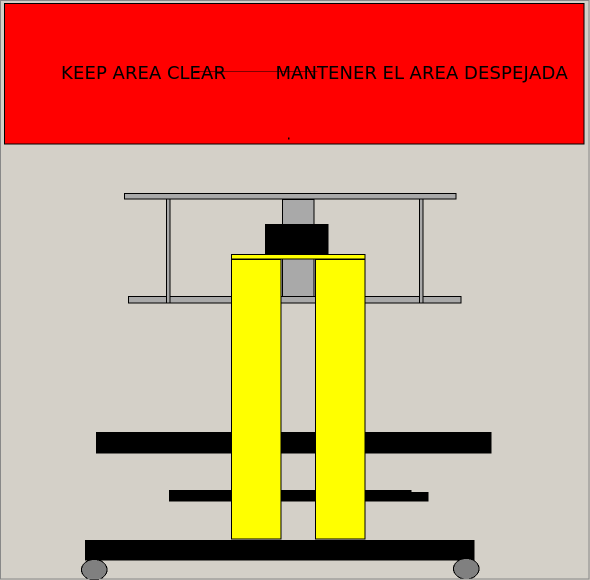
VISUALIZATION machineHomingScreen  // 590x580
    Rectangle (4,3 580x141)
    Rectangle (249,232 98x32), angle 90
    Rectangle (128,296 333x7)
    Rectangle (169,490 242x11), angle 25
    Rectangle (185,492 243x9), angle 336
    Rectangle (96,432 395x21)
    Rectangle (85,540 389x20)
    Rectangle (231,259 50x280)
    Rectangle (315,259 50x280)
    Ellipse (453,558 26x21)
    Ellipse (81,559 26x21)
    Rectangle (231,254 134x5)
    Rectangle (265,224 63x30)
    Rectangle (419,198 4x105)
    Rectangle (166,198 4x105)
    Rectangle (124,193 332x6)
    Label (18,48 251x50), "KEEP AREA CLEAR"
    Label (250,48 344x50), "MANTENER EL AREA DESPEJADA"
    Rectangle (288,138 1x0)
    Rectangle (194,71 123x0), angle 299
END_VISUALIZATION

(* stored: Version 1.1.0.1, ProductVersion 3.1.4024.15
   Visu machineHomingScreen: Id {564e3475-5ad8-4d8d-a8e6-0b3263008281} *)
